// SIMATIC S7-200 project (STEP 7-Micro/WIN), CPU 221 REL 01.10

SYMBOL_TABLE USER1
start_btn        I0.0
stop_btn         I0.1
s1               I0.2     // ra xi lanh C5
s2               I0.3     // cam bien tu A sang B
s3               I0.4     // cam bien thu 2
s4               I0.5     // cam bien vao day lap
s5               I0.6     // counter
s6               I0.7     // thu xi lanh C3
s7               I1.0     // ra xi lanh C3
s8               I1.1     // thu xi lanh C4
s9               I1.2     // giua xi lanh C4
s10              I1.3     // ra xi lanh C4
s12              I1.4     // day binh dinh luong
s14              I1.5     // day coc
C1_P             Q0.0     // rot vao binh dinh luong
C2_P             Q0.1     // mo binh dinh luong
C3_P             Q0.2     // day lap vao
C4_P             Q0.3     // hut nap chan khong
C5_P             Q0.4     // day lon tu A sang B
B_tai            Q0.5     // bang tai
END_SYMBOL_TABLE

ORGANIZATION_BLOCK MAIN:OB1
TITLE=PROGRAM COMMENTS
BEGIN
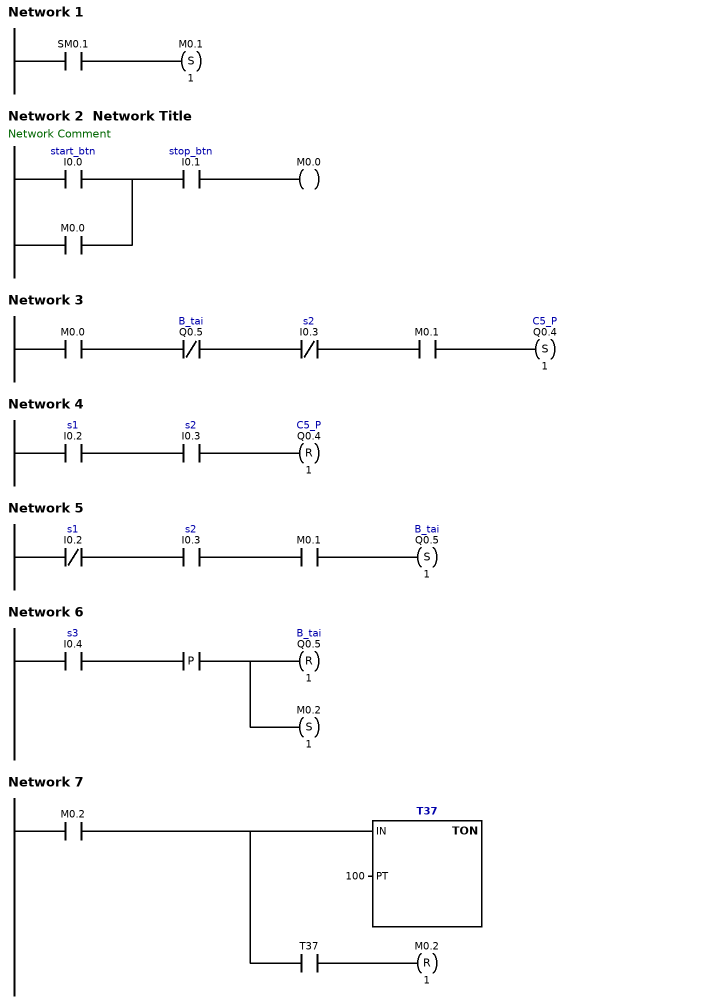
Network 1
// (network saved uncompiled; LAD cells follow)
// row 0: c0 -| |- SM0.1  c1 -(S) M0.1, 1
Network 2 // Network Title
// Network Comment
// (network saved uncompiled; LAD cells follow)
// row 0: c0 -| |- start_btn:I0.0 v  c1 -| |- stop_btn:I0.1  c2 -( ) M0.0
// row 1: c0 -| |- M0.0 ^
Network 3
// (network saved uncompiled; LAD cells follow)
// row 0: c0 -| |- M0.0  c1 -|/|- B_tai:Q0.5  c2 -|/|- s2:I0.3  c3 -| |- M0.1  c4 -(S) C5_P:Q0.4, 1
Network 4
// (network saved uncompiled; LAD cells follow)
// row 0: c0 -| |- s1:I0.2  c1 -| |- s2:I0.3  c2 -(R) C5_P:Q0.4, 1
Network 5
// (network saved uncompiled; LAD cells follow)
// row 0: c0 -|/|- s1:I0.2  c1 -| |- s2:I0.3  c2 -| |- M0.1  c3 -(S) B_tai:Q0.5, 1
Network 6
// (network saved uncompiled; LAD cells follow)
// row 0: c0 -| |- s3:I0.4  c1 -|P|-  v  c2 -(R) B_tai:Q0.5, 1
// row 1: c1 ^  c2 -(S) M0.2, 1
Network 7
// (network saved uncompiled; LAD cells follow)
// row 0: c0 -| |- M0.2  c1 -- v  c2 --  c3 [TON T37 IN:=power@row0, PT:=100]
// row 1: c1 ^v  c3 [box]
// row 2: c1 ^  c2 -| |- T37  c3 -(R) M0.2, 1
END_ORGANIZATION_BLOCK
